(* CODESYS project tcl_unittestlibrary.library
   Company: Red Rock Controls Limited
   Description: Support stand-alone test
   Version: 1.0.2.0
   Placeholder: tcl_UnitTestLibrary
   Author: Roger Christopher
   Title: tcl_UnitTestLibrary

Project tree, tasks and I/O mapping:
  libraries: Tc2_Standard, * (Beckhoff Automation GmbH); Tc2_System, * (Beckhoff Automation GmbH); Tc2_Utilities, * (Beckhoff Automation GmbH); Tc3_DynamicMemory, * (Beckhoff Automation GmbH); Tc3_Module, * (Beckhoff Automation GmbH); tcl_StringUtils, * (Red Rock Controls Limited)
  DUTs/
    data type ST_TestResult
  Functions/
  GVLs/
    global variables Parameters
  Unit Test Framework/
    Assertions/
      function F_Assert [ST]
      function block T_Assertion [ST]: Assert, AssertEquals_BLOB, AssertEquals_BOOL, AssertEquals_BYTE, AssertEquals_DINT, AssertEquals_DWORD, AssertEquals_INT, AssertEquals_INTERFACE, AssertEquals_LINT, AssertEquals_LREAL, AssertEquals_PVOID, AssertEquals_REAL, AssertEquals_STRING, AssertEquals_UDINT, AssertEquals_UINT, AssertEquals_ULINT, AssertEquals_WORD, AssertNotEquals_INTERFACE, AssertionFailed, AssertionMessage
    List Of Tests/
      interface I_ListOfTests: AddTest, Count, FindTestIndex, GetTest, SetTest, TestGroupName
      function block T_ListOfTests [ST]: AddTest, Clear, FB_exit, FB_init, FindTestIndex, GetTest, SetTest, Count, TestGroupName
      function block T_TestIterator [ST]: GetNext, HasMore, Initialise
    Test Runner/
      function block T_TestRunner [ST]: AddTest, Init, Start
    Unit Test/
      function F_LogResult [ST]
      interface I_UnitTest: Init, RunTest, TestGroupName, TestName
      function block T_UnitTestBase [ST]: FB_init_Old, Init, RunTest, SetTestName, TestGroupName, TestName
  Version/
    global variables Global_Version
*)

// DUTs/ST_TestResult
TYPE
    ST_TestResult :
    STRUCT
        TestCompleted : BOOL;
        TestFailed    : BOOL;
        FailMessage   : T_MaxString;
    END_STRUCT
END_TYPE

// GVLs/Parameters
VAR_GLOBAL CONSTANT
    MAX_TESTS : DINT := 200;
END_VAR

// Version/Global_Version
{attribute 'TcGenerated'}
{attribute 'no-analysis'}
{attribute 'linkalways'}
// This function has been automatically generated from the project information.
VAR_GLOBAL CONSTANT
	{attribute 'const_non_replaced'}
	stLibVersion_tcl_UnitTestLibrary : ST_LibVersion := (iMajor := 1, iMinor := 0, iBuild := 2, iRevision := 0, nFlags := 0, sVersion := '1.0.2.0');
END_VAR

// Unit Test Framework/Assertions/F_Assert
FUNCTION F_Assert : BOOL
VAR_INPUT
    Source       : T_MaxString;
    Expected     : ANY;
    Actual       : ANY;
    VariableName : T_MaxString;
END_VAR
VAR

END_VAR

IF Expected.TypeClass <> Actual.TypeClass THEN
    F_LogResult(Source := Source, Message := F_FormatStringEx1('Assertion failed on <%s> - TypeClass of expected and actual values differ',VariableName));
    RETURN;

ELSIF Expected.diSize <> Actual.diSize THEN
    F_LogResult(Source := Source, Message := F_FormatStringEx1('Assertion failed on <%s> - Sizes of expected and actual values differ',VariableName));
    RETURN;

ELSIF MEMCMP(pBuf1 := Expected.pValue, pBuf2 := Actual.pValue, n := DINT_TO_UDINT(Actual.diSize)) <> 0 THEN
    F_LogResult(Source := Source, Message := F_FormatStringEx1('Assertion failed on <%s> - Expected and actual values differ',VariableName));
    RETURN;
END_IF

F_Assert := TRUE;

END_FUNCTION

// Unit Test Framework/Unit Test/F_LogResult
FUNCTION F_LogResult : BOOL
VAR_INPUT
    Source  : T_MaxString;
    Message : T_MaxString;
END_VAR
VAR
END_VAR

ADSLOGSTR(msgCtrlMask := ADSLOG_MSGTYPE_STRING OR ADSLOG_MSGTYPE_ERROR OR ADSLOG_MSGTYPE_LOG,
          msgFmtStr   := F_FormatStringEx2('%s : %s', Source, Message),
          strArg      := '');

END_FUNCTION

// Unit Test Framework/Assertions/T_Assertion
FUNCTION_BLOCK T_Assertion
VAR_INPUT
END_VAR
VAR_OUTPUT
END_VAR
VAR
    _AssertionFailed  : BOOL;
    _AssertionMessage : T_MaxString;
    _ExpectedAsString : T_MaxString;
    _ActualAsString   : T_MaxString;
END_VAR

METHOD Assert
VAR_INPUT
    Caller           : T_MaxString;
    AssertionMessage : T_MaxString;
    Expected         : T_MaxString;
    Actual           : T_MaxString;
END_VAR
_AssertionFailed  := TRUE;
_AssertionMessage := F_FormatStringEx2('Assertion failed in %s - %s', Caller, AssertionMessage);
_ExpectedAsString := F_FormatStringEx1('  Expected = %s', Expected);
_ActualAsString   := F_FormatStringEx1('  Actual   = %s', Actual);
END_METHOD

METHOD AssertEquals_BLOB
VAR_INPUT
    Expected     : ANY;
    Actual       : ANY;
    VariableName : T_MaxString;
END_VAR
IF Expected.diSize <> Actual.diSize THEN
    _AssertionFailed  := TRUE;
    _AssertionMessage := F_FormatStringEx1('AssertEquals_BLOB failed in %s : Sizes differ', VariableName);

ELSIF Expected.TypeClass <> Actual.TypeClass THEN
    _AssertionFailed  := TRUE;
    _AssertionMessage := F_FormatStringEx1('AssertEquals_BLOB failed in %s: TypeClasses differ', VariableName);

ELSIF
    MEMCMP(pBuf1 := Expected.pValue, pBuf2 := Actual.pValue, n := DINT_TO_UDINT(Actual.diSize)) <> 0
THEN
    _AssertionFailed  := TRUE;
    _AssertionMessage := F_FormatStringEx1('AssertEquals_BLOB failed in %s: Contents differ', VariableName);
ELSE
    _AssertionFailed  := FALSE;
    _AssertionMessage := '';
END_IF
END_METHOD

METHOD AssertEquals_BOOL
VAR_INPUT
    Expected     : BOOL;
    Actual       : BOOL;
    VariableName : T_MaxString;
END_VAR
IF Expected <> Actual THEN
    _AssertionFailed  := TRUE;
    _AssertionMessage := F_FormatStringEx3('AssertEquals_BOOL failed : Variable "%s" =  %s, expected = %s', VariableName, BOOL_TO_STRING(Actual), BOOL_TO_STRING(Expected));
ELSE
    _AssertionFailed  := FALSE;
    _AssertionMessage := '';
END_IF
END_METHOD

METHOD AssertEquals_BYTE
VAR_INPUT
    Expected     : BYTE;
    Actual       : BYTE;
    VariableName : T_MaxString;
END_VAR
IF Expected <> Actual THEN
    _AssertionFailed  := TRUE;
    _AssertionMessage := F_FormatString3('AssertEquals_BYTE failed : Variable "%s" =  %d, expected = %d', F_STRING(VariableName), F_BYTE(Actual), F_BYTE(Expected));
ELSE
    _AssertionFailed  := FALSE;
    _AssertionMessage := '';
END_IF
END_METHOD

METHOD AssertEquals_DINT
VAR_INPUT
    Expected     : DINT;
    Actual       : DINT;
    VariableName : T_MaxString;
END_VAR
IF Expected <> Actual THEN
    _AssertionFailed  := TRUE;
    _AssertionMessage := F_FormatString3('AssertEquals_DINT failed : Variable "%s" =  %d, expected = %d', F_STRING(VariableName), F_DINT(Actual), F_DINT(Expected));
ELSE
    _AssertionFailed  := FALSE;
    _AssertionMessage := '';
END_IF
END_METHOD

METHOD AssertEquals_DWORD
VAR_INPUT
    Expected     : DWORD;
    Actual       : DWORD;
    VariableName : T_MaxString;
END_VAR
IF Expected <> Actual THEN
    _AssertionFailed  := TRUE;
    _AssertionMessage := F_FormatString3('AssertEquals_DWORD failed : Variable "%s" =  %d, expected = %d', F_STRING(VariableName), F_DWORD(Actual), F_DWORD(Expected));
ELSE
    _AssertionFailed  := FALSE;
    _AssertionMessage := '';
END_IF
END_METHOD

METHOD AssertEquals_INT
VAR_INPUT
    Expected     : INT;
    Actual       : INT;
    VariableName : T_MaxString;
END_VAR
IF Expected <> Actual THEN
    _AssertionFailed  := TRUE;
    _AssertionMessage := F_FormatString3('AssertEquals_INT failed : Variable "%s" =  %d, expected = %d', F_STRING(VariableName), F_INT(Actual), F_INT(Expected));
ELSE
    _AssertionFailed  := FALSE;
    _AssertionMessage := '';
END_IF
END_METHOD

METHOD AssertEquals_INTERFACE
VAR_INPUT
    Expected     : __SYSTEM.IQueryInterface;
    Actual       : __SYSTEM.IQueryInterface;
    VariableName : T_MaxString;
END_VAR
IF Expected <> Actual THEN
    _AssertionFailed  := TRUE;
    _AssertionMessage := F_FormatString1('AssertEquals_INTERFACE failed : Variable "%s"', F_STRING(VariableName));
ELSE
    _AssertionFailed  := FALSE;
    _AssertionMessage := '';
END_IF
END_METHOD

METHOD AssertEquals_LINT
VAR_INPUT
    Expected     : LINT;
    Actual       : LINT;
    VariableName : T_MaxString;
END_VAR
IF Expected <> Actual THEN
    _AssertionFailed  := TRUE;
    _AssertionMessage := F_FormatString3('AssertEquals_LINT failed : Variable "%s" =  %d, expected = %d', F_STRING(VariableName), F_LINT(Actual), F_LINT(Expected));
ELSE
    _AssertionFailed  := FALSE;
    _AssertionMessage := '';
END_IF
END_METHOD

METHOD AssertEquals_LREAL
VAR_INPUT
    Expected     : LREAL;
    Actual       : LREAL;
    Delta        : LREAL;
    VariableName : T_MaxString;
END_VAR
IF ABS(Expected - Actual) > Delta THEN
    _AssertionFailed  := TRUE;
    _AssertionMessage := F_FormatString3('AssertEquals_LREAL failed : Variable "%s" =  %f, expected = %f', F_STRING(VariableName), F_LREAL(Actual), F_LREAL(Expected));
ELSE
    _AssertionFailed  := FALSE;
    _AssertionMessage := '';
END_IF
END_METHOD

METHOD AssertEquals_PVOID
VAR_INPUT
    Expected     : PVOID;
    Actual       : PVOID;
    VariableName : T_MaxString;
END_VAR
IF Expected <> Actual THEN
    _AssertionFailed  := TRUE;
    _AssertionMessage := F_FormatString1('AssertEquals_PVOID failed : Variable "%s"', F_STRING(VariableName));
ELSE
    _AssertionFailed  := FALSE;
    _AssertionMessage := '';
END_IF
END_METHOD

METHOD AssertEquals_REAL
VAR_INPUT
    Expected     : REAL;
    Actual       : REAL;
    Delta        : REAL;
    VariableName : T_MaxString;
END_VAR
IF ABS(Expected - Actual) > Delta THEN
    _AssertionFailed  := TRUE;
    _AssertionMessage := F_FormatString3('AssertEquals_REAL failed : Variable "%s" =  %f, expected = %f', F_STRING(VariableName), F_REAL(Actual), F_REAL(Expected));
ELSE
    _AssertionFailed  := FALSE;
    _AssertionMessage := '';
END_IF
END_METHOD

METHOD AssertEquals_STRING
VAR_INPUT
    Expected     : T_MaxString;
    Actual       : T_MaxString;
    VariableName : T_MaxString;
END_VAR
IF Expected <> Actual THEN
    _AssertionFailed  := TRUE;
    _AssertionMessage := F_FormatString3('AssertEquals_STRING failed : Variable "%s" =  %s, expected = %s', F_STRING(VariableName), F_STRING(Actual), F_STRING(Expected));
ELSE
    _AssertionFailed  := FALSE;
    _AssertionMessage := '';
    _ExpectedAsString := '';
    _ActualAsString   := '';
END_IF
END_METHOD

METHOD AssertEquals_UDINT
VAR_INPUT
    Expected     : UDINT;
    Actual       : UDINT;
    VariableName : T_MaxString;
END_VAR
IF Expected <> Actual THEN
    _AssertionFailed  := TRUE;
    _AssertionMessage := F_FormatString3('AssertEquals_UDINT failed : Variable "%s" =  %d, expected = %d', F_STRING(VariableName), F_UDINT(Actual), F_UDINT(Expected));
ELSE
    _AssertionFailed  := FALSE;
    _AssertionMessage := '';
END_IF
END_METHOD

METHOD AssertEquals_UINT
VAR_INPUT
    Expected     : UINT;
    Actual       : UINT;
    VariableName : T_MaxString;
END_VAR
IF Expected <> Actual THEN
    _AssertionFailed  := TRUE;
    _AssertionMessage := F_FormatString3('AssertEquals_UINT failed : Variable "%s" =  %d, expected = %d', F_STRING(VariableName), F_UINT(Actual), F_UINT(Expected));
ELSE
    _AssertionFailed  := FALSE;
    _AssertionMessage := '';
END_IF
END_METHOD

METHOD AssertEquals_ULINT
VAR_INPUT
    Expected     : ULINT;
    Actual       : ULINT;
    VariableName : T_MaxString;
END_VAR
IF Expected <> Actual THEN
    _AssertionFailed  := TRUE;
    _AssertionMessage := F_FormatString3('AssertEquals_ULINT failed : Variable "%s" =  %d, expected = %d', F_STRING(VariableName), F_ULINT(Actual), F_ULINT(Expected));
ELSE
    _AssertionFailed  := FALSE;
    _AssertionMessage := '';
END_IF
END_METHOD

METHOD AssertEquals_WORD
VAR_INPUT
    Expected     : WORD;
    Actual       : WORD;
    VariableName : T_MaxString;
END_VAR
IF Expected <> Actual THEN
    _AssertionFailed  := TRUE;
    _AssertionMessage := F_FormatString3('AssertEquals_WORD failed : Variable "%s" =  %d, expected = %d', F_STRING(VariableName), F_WORD(Actual), F_WORD(Expected));
ELSE
    _AssertionFailed  := FALSE;
    _AssertionMessage := '';
END_IF
END_METHOD

METHOD AssertNotEquals_INTERFACE
VAR_INPUT
    Expected     : __SYSTEM.IQueryInterface;
    Actual       : __SYSTEM.IQueryInterface;
    VariableName : T_MaxString;
END_VAR
IF Expected = Actual THEN
    _AssertionFailed  := TRUE;
    _AssertionMessage := F_FormatString1('AssertNotEquals_INTERFACE failed : Variable "%s"', F_STRING(VariableName));
ELSE
    _AssertionFailed  := FALSE;
    _AssertionMessage := '';
END_IF
END_METHOD

PROPERTY AssertionFailed : BOOL
GET
AssertionFailed := _AssertionFailed;
END_GET
END_PROPERTY

PROPERTY AssertionMessage : T_MaxString
GET
AssertionMessage := _AssertionMessage;
END_GET
END_PROPERTY

END_FUNCTION_BLOCK

// Unit Test Framework/List Of Tests/I_ListOfTests
INTERFACE I_ListOfTests

METHOD AddTest
VAR_INPUT
    Test : I_UnitTest;
END_VAR
END_METHOD

PROPERTY Count : DINT
GET
END_GET
END_PROPERTY

METHOD FindTestIndex : DINT
VAR_INPUT
	Test : I_UnitTest;
END_VAR
END_METHOD

METHOD GetTest : I_UnitTest
VAR_INPUT
    Index : DINT;
END_VAR
END_METHOD

METHOD SetTest : I_UnitTest
VAR_INPUT
    Test : I_UnitTest;
    Index : DINT;
END_VAR
END_METHOD

PROPERTY TestGroupName : T_MaxString
GET
END_GET
END_PROPERTY

END_INTERFACE

// Unit Test Framework/Unit Test/I_UnitTest
INTERFACE I_UnitTest EXTENDS __SYSTEM.IQueryInterface

METHOD Init : BOOL
VAR_INPUT
END_VAR
END_METHOD

METHOD FINAL RunTest
VAR_OUTPUT
    TestCompleted : BOOL;
    TestFailed    : BOOL;
END_VAR
END_METHOD

PROPERTY TestGroupName : T_MaxString
GET
END_GET
END_PROPERTY

PROPERTY TestName : T_MaxString
GET
END_GET
END_PROPERTY

END_INTERFACE

// Unit Test Framework/List Of Tests/T_ListOfTests
FUNCTION_BLOCK T_ListOfTests IMPLEMENTS I_ListOfTests
VAR
    _TestGroupName       : T_MaxString;
    Buffer               : FB_DynMem_Buffer(ipMemMan := DynamicMemoryManager);
    DynamicMemoryManager : FB_DynMem_Manager;
    pTest                : POINTER TO I_UnitTest;
    _Count               : DINT;
    Capacity             : DINT;
	
	FindTestResult : DINT;
END_VAR

METHOD AddTest
VAR_INPUT
    Test : I_UnitTest;
END_VAR
IF _Count = Capacity THEN
    Capacity := Capacity * 2;
    Buffer.Resize(nSize     := DINT_TO_UDINT(Capacity) * SIZEOF(PVOID),
                  bPreserve := TRUE,
                  bReset    := FALSE);

    pTest := Buffer.pBuffer;
END_IF

pTest[_Count] := Test;
_Count        := _Count + 1;
END_METHOD

METHOD Clear
VAR_INPUT
END_VAR
Buffer.Clear();
_Count := 0;
END_METHOD

METHOD FB_exit : BOOL
VAR_INPUT
    bInCopyCode : BOOL; // if TRUE, the exit method is called for exiting an instance that is copied afterwards (online change).
END_VAR
IF NOT bInCopyCode THEN
    Buffer.DeleteBuffer();
    pTest := 0;
END_IF
END_METHOD

METHOD FB_init : BOOL
VAR_INPUT
    bInitRetains  : BOOL; // if TRUE, the retain variables are initialized (warm start / cold start)
    bInCopyCode   : BOOL; // if TRUE, the instance afterwards gets moved into the copy code (online change)
    Capacity      : DINT;
END_VAR
Buffer.CreateBuffer(nSize  := DINT_TO_UDINT(Capacity) * SIZEOF(PVOID),
                    bReset := TRUE);

pTest                := Buffer.pBuffer;
THIS^.Capacity       := Capacity;
END_METHOD

METHOD FindTestIndex : DINT
VAR_INPUT
	Test : I_UnitTest;
END_VAR
VAR
	NextTest : I_UnitTest;
	i : DINT;
END_VAR
FOR i := 0 TO _Count - 1 DO
	NextTest := GetTest(i);
	IF NextTest = Test THEN
		FindTestIndex := i;
		FindTestResult := i;
		RETURN;
	END_IF
END_FOR
FindTestIndex := -1;
FindTestResult := -1;
END_METHOD

METHOD GetTest : I_UnitTest
VAR_INPUT
    Index : DINT;
END_VAR
IF Index < _Count AND Index >= 0 THEN
    GetTest := pTest[Index];
END_IF
END_METHOD

METHOD SetTest : I_UnitTest
VAR_INPUT
    Test : I_UnitTest;
    Index : DINT;
END_VAR
IF Index < _Count AND Index >= 0 THEN
    pTest[Index] := Test;
END_IF
END_METHOD

PROPERTY Count : DINT
GET
Count := _Count;
END_GET
END_PROPERTY

PROPERTY TestGroupName : T_MaxString
GET
TestGroupName := _TestGroupName;
END_GET
END_PROPERTY

END_FUNCTION_BLOCK

// Unit Test Framework/List Of Tests/T_TestIterator
FUNCTION_BLOCK T_TestIterator
VAR_INPUT
END_VAR
VAR_OUTPUT
END_VAR
VAR
    List  : I_ListOfTests;
    Index : DINT;
END_VAR

METHOD GetNext : I_UnitTest
VAR_INPUT
END_VAR
IF List <> 0 AND_THEN HasMore() THEN
    GetNext := List.GetTest(Index);
    Index   := Index + 1;
END_IF
END_METHOD

METHOD HasMore : BOOL
VAR_INPUT
END_VAR
HasMore := List <> 0 AND_THEN (Index < List.Count and List.Count > 0);
END_METHOD

METHOD Initialise : BOOL
VAR_INPUT
    List         : I_ListOfTests;
END_VAR
THIS^.List := List;
Index      := 0;
END_METHOD

END_FUNCTION_BLOCK

// Unit Test Framework/Test Runner/T_TestRunner
FUNCTION_BLOCK T_TestRunner
VAR
    State : (
        sInit,
        sGetTest,
        sRunTest,
        sCheckResults
    );
    ResultsSummary          : T_MaxString;
    PassedTestsCount        : DINT;
    FailedTestsCount        : DINT;
    TestList                : T_ListOfTests(Capacity := 50);
    TestIterator            : T_TestIterator;
    CurrentTest             : I_UnitTest;

	RunTests : BOOL;
    TestFailed    : BOOL;
    TestCompleted : BOOL;
END_VAR

CASE State OF
    sInit:
        IF RunTests THEN
            RunTests := FALSE;
            TestIterator.Initialise(TestList);
            ResultsSummary   := '';
            FailedTestsCount := 0;
            PassedTestsCount := 0;
            State            := sGetTest;
        END_IF

    sGetTest:
        IF TestIterator.HasMore() THEN
            CurrentTest := TestIterator.GetNext();
            CurrentTest.Init();
            State := sRunTest;
        ELSE
            CurrentTest := 0;
            State       := sCheckResults;
        END_IF

    sRunTest:
        CurrentTest.RunTest(TestCompleted => TestCompleted,
                            TestFailed    => TestFailed);

        IF TestCompleted THEN
            IF TestFailed THEN
                FailedTestsCount := FailedTestsCount + 1;
            ELSE
                PassedTestsCount := PassedTestsCount + 1;
            END_IF
            State := sGetTest;
        END_IF

    sCheckResults:
        ResultsSummary := F_FormatString2('%d Tests Passed, %d Tests Failed',
                                          F_DINT(PassedTestsCount),
                                          F_DINT(FailedTestsCount));

        F_LogResult(Source  := 'Unit Test Runner',
                    Message := F_FormatString2('%d Tests Passed, %d Tests Failed',
                                               F_DINT(PassedTestsCount),
                                               F_DINT(FailedTestsCount)));
        State := sInit;

END_CASE

METHOD AddTest
VAR_INPUT
    UnitTest : I_UnitTest;
END_VAR
TestList.AddTest(UnitTest);
END_METHOD

METHOD Init
VAR_INPUT
END_VAR
TestList.Clear();
END_METHOD

METHOD Start
VAR_INPUT
END_VAR
RunTests := TRUE;
END_METHOD

END_FUNCTION_BLOCK

// Unit Test Framework/Unit Test/T_UnitTestBase
{attribute 'reflection'}
{attribute 'hide_all_locals'}
FUNCTION_BLOCK ABSTRACT T_UnitTestBase IMPLEMENTS I_UnitTest
VAR_INPUT
END_VAR
VAR_OUTPUT
END_VAR
VAR
    {attribute 'instance-path'}
    {attribute 'no_init'}
    _InstanceName  : T_MaxString; // Automatically initialised with the full name of the instance
    _TestGroupName : T_MaxString;
    _TestName      : T_MaxString;
    _TestResult    : ST_TestResult;

    State : INT;        // for general use during test...
END_VAR

METHOD FB_init_Old : BOOL
VAR_INPUT
    bInitRetains : BOOL; // if TRUE, the retain variables are initialized (warm start / cold start)
    bInCopyCode  : BOOL; // if TRUE, the instance afterwards gets moved into the copy code (online change)
	ListOfTests : I_ListOfTests;
END_VAR
VAR
	Index : DINT;
END_VAR
THIS^.SetTestName();
IF ListOfTests <> 0 THEN
    THIS^._TestGroupName := ListOfTests.TestGroupName;
	
	IF NOT bInCopyCode THEN //not online change
        ListOfTests.AddTest(Test := THIS^);
	END_IF
	
END_IF
END_METHOD

METHOD ABSTRACT Init : BOOL
END_METHOD

METHOD ABSTRACT RunTest
VAR_OUTPUT
    TestCompleted : BOOL;
    TestFailed    : BOOL;
END_VAR
END_METHOD

METHOD PRIVATE SetTestName
VAR
    StringSplitter : T_StringSplitter;
END_VAR
StringSplitter.Init(Str    := _InstanceName,
                    Delim1 := '.',
                    Delim2 := '');

WHILE StringSplitter.HasMore() DO
    _TestName := StringSplitter.GetNext(); // to get last sub-section
END_WHILE
END_METHOD

PROPERTY TestGroupName : T_MaxString
GET
TestGroupName := _TestGroupName;
END_GET
END_PROPERTY

PROPERTY TestName : T_MaxString
GET
TestName := _TestName;
END_GET
END_PROPERTY

END_FUNCTION_BLOCK
